// TIA Portal V20 export
TYPE "UDT_EmptyPosition"
   STRUCT
      Presence : "UDT_PartPresence";
      States : "UDT_PartStates";
   END_STRUCT;
END_TYPE
